PROGRAM MP_1_Y100
VAR
	CompareOutput100_00: CMP_OC_DW;
	CompareOutput100_01: CMP_OC_DW;
	CompareOutput100_02: CMP_OC_DW;
	CompareOutput100_03: CMP_OC_DW;
	CompareOutput100_04: CMP_OC_DW;
	CompareOutput100_05: CMP_OC_DW;
	CompareOutput100_06: CMP_OC_DW;
	CompareOutput100_07: CMP_OC_DW;
	CompareOutput100_08: CMP_OC_DW;
	CompareOutput100_09: CMP_OC_DW;
	CompareOutput100_10: CMP_OC_DW;
	CompareOutput100_11: CMP_OC_DW;
	CompareOutput100_12: CMP_OC_DW;
	CompareOutput100_13: CMP_OC_DW;
	CompareOutput100_14: CMP_OC_DW;
	CompareOutput100_15: CMP_OC_DW;

	tEStopDelayOnTimer: TON;
	tHeaterPIDResetDelayOnTimer: TON;
END_VAR

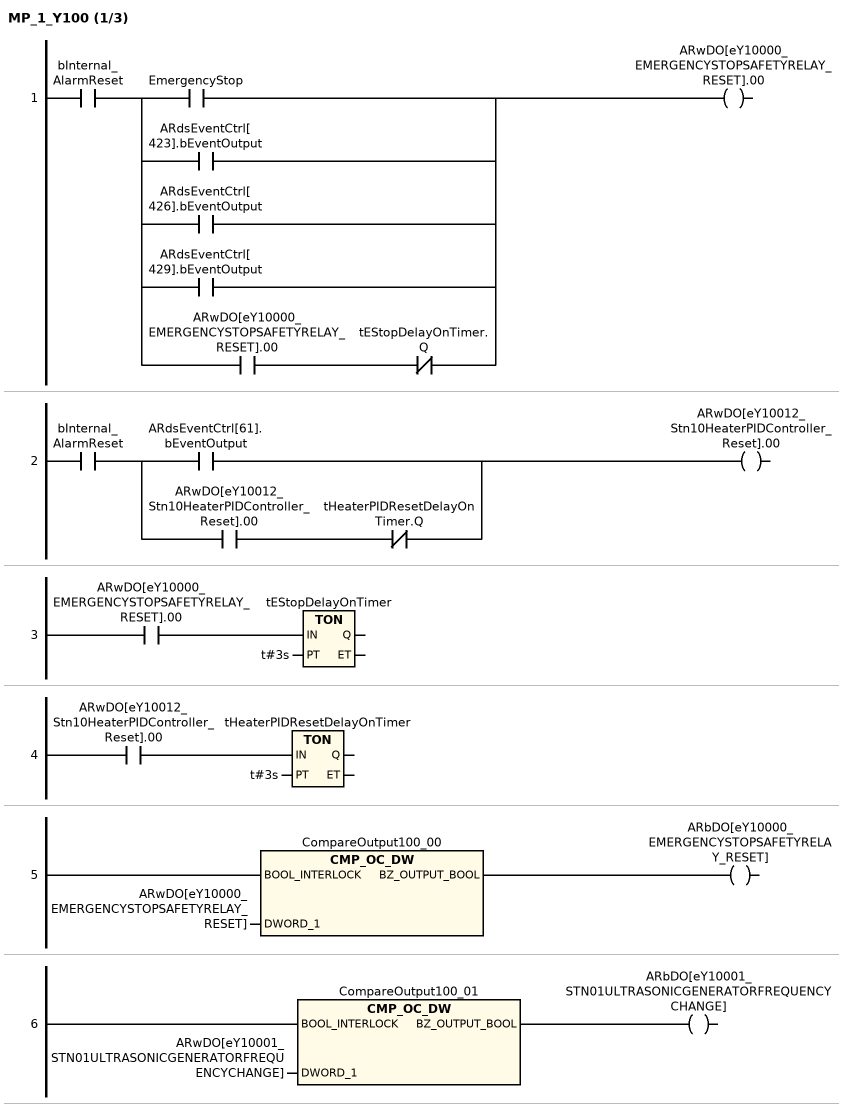
// NETWORK 1
ARwDO[eY10000_EMERGENCYSTOPSAFETYRELAY_RESET].00 := bInternal_AlarmReset AND (EmergencyStop OR ARdsEventCtrl[423].bEventOutput OR ARdsEventCtrl[426].bEventOutput OR ARdsEventCtrl[429].bEventOutput OR ARwDO[eY10000_EMERGENCYSTOPSAFETYRELAY_RESET].00 AND NOT tEStopDelayOnTimer.Q);

// NETWORK 2
ARwDO[eY10012_Stn10HeaterPIDController_Reset].00 := bInternal_AlarmReset AND (ARdsEventCtrl[61].bEventOutput OR ARwDO[eY10012_Stn10HeaterPIDController_Reset].00 AND NOT tHeaterPIDResetDelayOnTimer.Q);

// NETWORK 3
tEStopDelayOnTimer(IN := ARwDO[eY10000_EMERGENCYSTOPSAFETYRELAY_RESET].00, PT := t#3s); // TON

// NETWORK 4
tHeaterPIDResetDelayOnTimer(IN := ARwDO[eY10012_Stn10HeaterPIDController_Reset].00, PT := t#3s); // TON

// NETWORK 5
CompareOutput100_00(BOOL_INTERLOCK := TRUE, DWORD_1 := ARwDO[eY10000_EMERGENCYSTOPSAFETYRELAY_RESET]); // CMP_OC_DW
ARbDO[eY10000_EMERGENCYSTOPSAFETYRELAY_RESET] := CompareOutput100_00.BZ_OUTPUT_BOOL;

// NETWORK 6
CompareOutput100_01(BOOL_INTERLOCK := TRUE, DWORD_1 := ARwDO[eY10001_STN01ULTRASONICGENERATORFREQUENCYCHANGE]); // CMP_OC_DW
ARbDO[eY10001_STN01ULTRASONICGENERATORFREQUENCYCHANGE] := CompareOutput100_01.BZ_OUTPUT_BOOL;

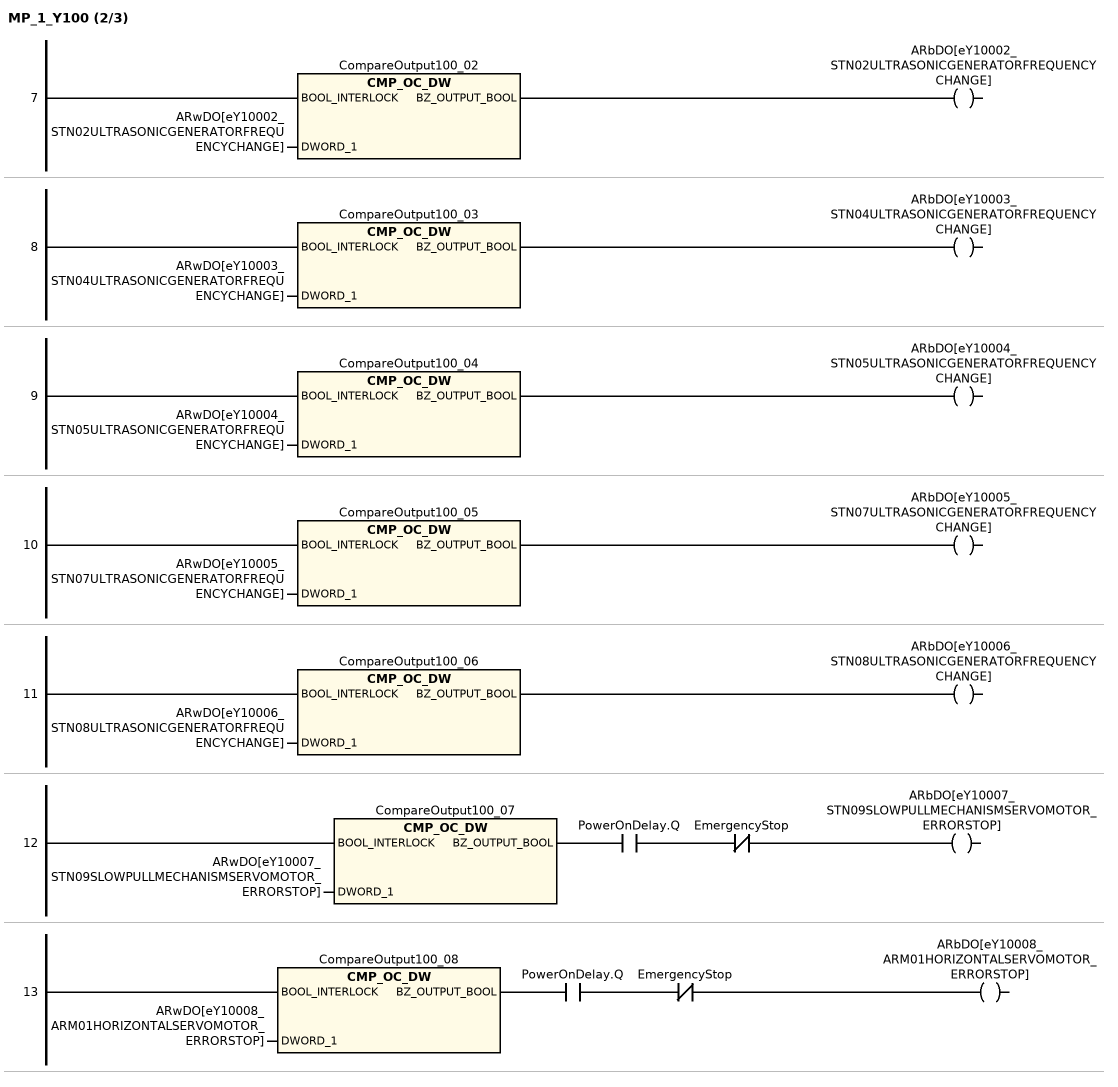
// NETWORK 7
CompareOutput100_02(BOOL_INTERLOCK := TRUE, DWORD_1 := ARwDO[eY10002_STN02ULTRASONICGENERATORFREQUENCYCHANGE]); // CMP_OC_DW
ARbDO[eY10002_STN02ULTRASONICGENERATORFREQUENCYCHANGE] := CompareOutput100_02.BZ_OUTPUT_BOOL;

// NETWORK 8
CompareOutput100_03(BOOL_INTERLOCK := TRUE, DWORD_1 := ARwDO[eY10003_STN04ULTRASONICGENERATORFREQUENCYCHANGE]); // CMP_OC_DW
ARbDO[eY10003_STN04ULTRASONICGENERATORFREQUENCYCHANGE] := CompareOutput100_03.BZ_OUTPUT_BOOL;

// NETWORK 9
CompareOutput100_04(BOOL_INTERLOCK := TRUE, DWORD_1 := ARwDO[eY10004_STN05ULTRASONICGENERATORFREQUENCYCHANGE]); // CMP_OC_DW
ARbDO[eY10004_STN05ULTRASONICGENERATORFREQUENCYCHANGE] := CompareOutput100_04.BZ_OUTPUT_BOOL;

// NETWORK 10
CompareOutput100_05(BOOL_INTERLOCK := TRUE, DWORD_1 := ARwDO[eY10005_STN07ULTRASONICGENERATORFREQUENCYCHANGE]); // CMP_OC_DW
ARbDO[eY10005_STN07ULTRASONICGENERATORFREQUENCYCHANGE] := CompareOutput100_05.BZ_OUTPUT_BOOL;

// NETWORK 11
CompareOutput100_06(BOOL_INTERLOCK := TRUE, DWORD_1 := ARwDO[eY10006_STN08ULTRASONICGENERATORFREQUENCYCHANGE]); // CMP_OC_DW
ARbDO[eY10006_STN08ULTRASONICGENERATORFREQUENCYCHANGE] := CompareOutput100_06.BZ_OUTPUT_BOOL;

// NETWORK 12
CompareOutput100_07(BOOL_INTERLOCK := TRUE, DWORD_1 := ARwDO[eY10007_STN09SLOWPULLMECHANISMSERVOMOTOR_ERRORSTOP]); // CMP_OC_DW
ARbDO[eY10007_STN09SLOWPULLMECHANISMSERVOMOTOR_ERRORSTOP] := CompareOutput100_07.BZ_OUTPUT_BOOL AND PowerOnDelay.Q AND NOT EmergencyStop;

// NETWORK 13
CompareOutput100_08(BOOL_INTERLOCK := TRUE, DWORD_1 := ARwDO[eY10008_ARM01HORIZONTALSERVOMOTOR_ERRORSTOP]); // CMP_OC_DW
ARbDO[eY10008_ARM01HORIZONTALSERVOMOTOR_ERRORSTOP] := CompareOutput100_08.BZ_OUTPUT_BOOL AND PowerOnDelay.Q AND NOT EmergencyStop;

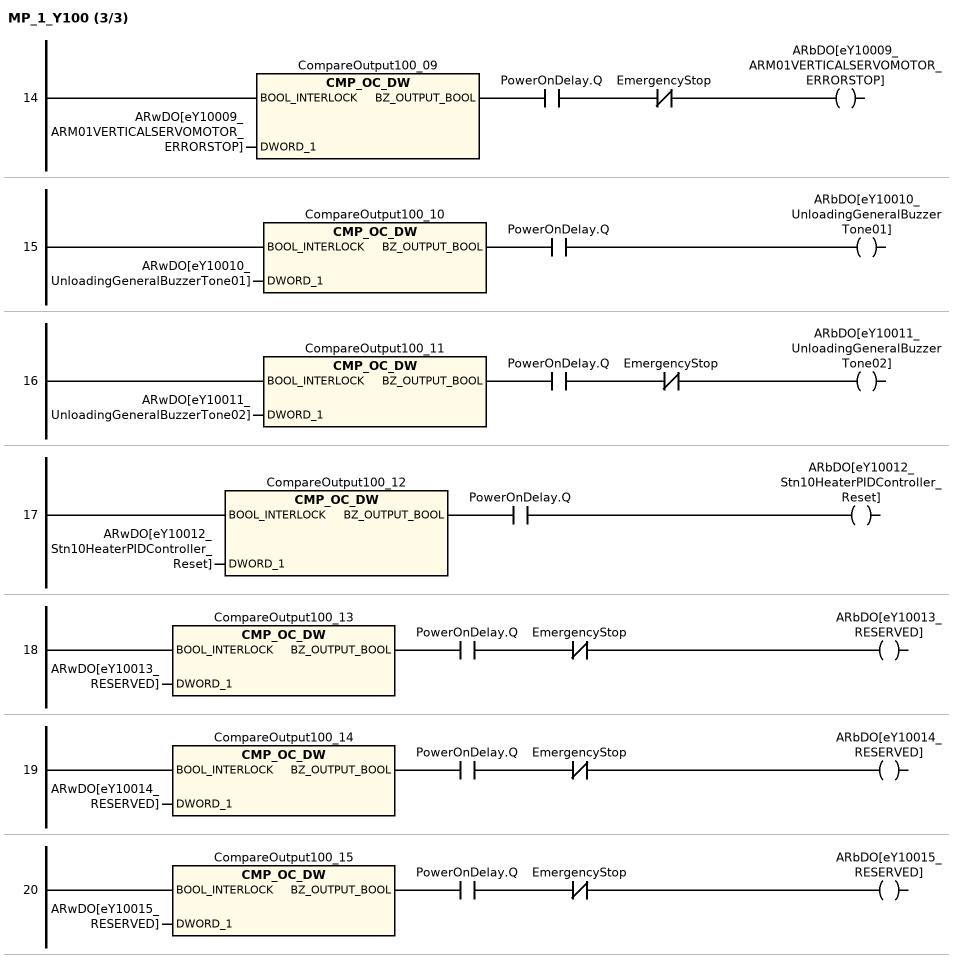
// NETWORK 14
CompareOutput100_09(BOOL_INTERLOCK := TRUE, DWORD_1 := ARwDO[eY10009_ARM01VERTICALSERVOMOTOR_ERRORSTOP]); // CMP_OC_DW
ARbDO[eY10009_ARM01VERTICALSERVOMOTOR_ERRORSTOP] := CompareOutput100_09.BZ_OUTPUT_BOOL AND PowerOnDelay.Q AND NOT EmergencyStop;

// NETWORK 15
CompareOutput100_10(BOOL_INTERLOCK := TRUE, DWORD_1 := ARwDO[eY10010_UnloadingGeneralBuzzerTone01]); // CMP_OC_DW
ARbDO[eY10010_UnloadingGeneralBuzzerTone01] := CompareOutput100_10.BZ_OUTPUT_BOOL AND PowerOnDelay.Q;

// NETWORK 16
CompareOutput100_11(BOOL_INTERLOCK := TRUE, DWORD_1 := ARwDO[eY10011_UnloadingGeneralBuzzerTone02]); // CMP_OC_DW
ARbDO[eY10011_UnloadingGeneralBuzzerTone02] := CompareOutput100_11.BZ_OUTPUT_BOOL AND PowerOnDelay.Q AND NOT EmergencyStop;

// NETWORK 17
CompareOutput100_12(BOOL_INTERLOCK := TRUE, DWORD_1 := ARwDO[eY10012_Stn10HeaterPIDController_Reset]); // CMP_OC_DW
ARbDO[eY10012_Stn10HeaterPIDController_Reset] := CompareOutput100_12.BZ_OUTPUT_BOOL AND PowerOnDelay.Q;

// NETWORK 18
CompareOutput100_13(BOOL_INTERLOCK := TRUE, DWORD_1 := ARwDO[eY10013_RESERVED]); // CMP_OC_DW
ARbDO[eY10013_RESERVED] := CompareOutput100_13.BZ_OUTPUT_BOOL AND PowerOnDelay.Q AND NOT EmergencyStop;

// NETWORK 19
CompareOutput100_14(BOOL_INTERLOCK := TRUE, DWORD_1 := ARwDO[eY10014_RESERVED]); // CMP_OC_DW
ARbDO[eY10014_RESERVED] := CompareOutput100_14.BZ_OUTPUT_BOOL AND PowerOnDelay.Q AND NOT EmergencyStop;

// NETWORK 20
CompareOutput100_15(BOOL_INTERLOCK := TRUE, DWORD_1 := ARwDO[eY10015_RESERVED]); // CMP_OC_DW
ARbDO[eY10015_RESERVED] := CompareOutput100_15.BZ_OUTPUT_BOOL AND PowerOnDelay.Q AND NOT EmergencyStop;

END_PROGRAM

(* stored: Version 1.1.0.1, ProductVersion 3.1.4024.11
   POU MP_1_Y100: Id {d348cdfd-b6bc-45c6-bc4e-9bec7e0562f8}, SpecialFunc None *)
